  (*-- TRANSITION --------------------------------------------------------------------------------------------------------------*)
  IF (_CreateDir.bBusy = FALSE)
  THEN
    (*-- folder created => continue -----------------------------------------------------*)
    IF ( _CreateDir.bError = FALSE )
    THEN
      _WriteState:= E_TraceWriteStates.ScanFileStart;
      (*-- trace it -------------------------------------------------*)
// example: '11-000-0000-00-0, new folder created,  folder = D:/Traces/1979-01-09/'
      _Text:= '';
      _Text:= CONCAT(_Text, F_AddDividerToSisString(SubsystemRegistry.SubsystemName) );
      _Text:= CONCAT(_Text, ',  new folder created');
      _Text:= CONCAT(_Text, DebugTextBlocks.FOLDER);
      _Text:= CONCAT(_Text, _CreateDir.sPathName);
      Put( MsgType := E_DebugMsgType.INFO,
           Instance:= ADR(_Instance),
           Text    := ADR(_Text)  );
    (*-- folder already exists ----------------------------------------------------------*)
    ELSIF (    ( _CreateDir.nErrId = 16#070C )     // ADSERR_DEVICE_NOTFOUND
            OR ( _CreateDir.nErrId = 16#0723 )  )  // ADSERR_DEVICE_ACCESSDENIED
    THEN                                           // BKF-Flick: Änderung der ReturnCodes ab 4022.20
      _WriteState:= E_TraceWriteStates.ScanFileStart;
    (*-- error --------------------------------------------------------------------------*)
    ELSE
      _WriteState:= E_TraceWriteStates.Error;
    END_IF
  END_IF




(********************************************************************************************************************************)
(** prepare folder scan for existing files **************************************************************************************)
E_TraceWriteStates.ScanFileStart:
  (*-- ENTRY -------------------------------------------------------------------------------------------------------------------*)
  IF (_WriteStateLast <> _WriteState)
  THEN
    _WriteStateLast:= _WriteState;
    _WriteTime     := F_GetTimeMsTick();
    (*-----------------------------------------------------------------------------------*)
    _FileIndex     := 1;  (* Filenummerierung beginnt bei Eins *)
    _FileCheck.eCmd:= eEnumCmd_First;
  END_IF

  (*-- ACTION ------------------------------------------------------------------------------------------------------------------*)

  (*-- TRANSITION --------------------------------------------------------------------------------------------------------------*)
    _WriteState:= E_TraceWriteStates.ScanFileExists;




(********************************************************************************************************************************)
(** scan folder to check if files exist? ****************************************************************************************)
E_TraceWriteStates.ScanFileExists:
  (*-- ENTRY -------------------------------------------------------------------------------------------------------------------*)
  IF (_WriteStateLast <> _WriteState)
  THEN
    _WriteStateLast:= _WriteState;
    _WriteTime     := F_GetTimeMsTick();
    (*-- build file name with _FileIndex ------------------------------------------------*)
{warning disable C0139}
    M_BuildFileName();    _WriteFileName;
{warning restore C0139}
   (*-----------------------------------------------------------------------------------*)
    _FileCheck( bExecute:= FALSE );
    _FileCheck.sNetID   := '';  // local
//  _FileCheck.eCmd;   // maintain this value here 
    _FileCheck.bExecute := TRUE;
    _FileCheck.tTimeout := Tc2_System.DEFAULT_ADS_TIMEOUT;
    (*-----------------------------------------------------------------------------------*)
    DestStart:= ADR(_FileCheck.sPathName);
    DestEnd  := ADR(_FileCheck.sPathName) + SIZEOF(_FileCheck.sPathName);
    DestStart:= F_StringCopy( DestStart:= DestStart,  DestEnd:= DestEnd,  Source:= ADR(_WritePath)  );
    DestStart:= F_StringCopy( DestStart:= DestStart,  DestEnd:= DestEnd,  Source:= ADR(_WriteFileName)  );
  END_IF

  (*-- ACTION ------------------------------------------------------------------------------------------------------------------*)
  _FileCheck();

  (*-- TRANSITION --------------------------------------------------------------------------------------------------------------*)
  IF (_FileCheck.bBusy = FALSE)
  THEN
    _FileCheck.eCmd:= E_EnumCmdType.eEnumCmd_Next;
    (*-- error --------------------------------------------------------------------------*)
    IF ( _FileCheck.bError = TRUE )
    THEN
      _WriteState:= E_TraceWriteStates.Error;
    (*-- index does not exist => create & use -------------------------------------------*)
    ELSIF ( _FileCheck.bEOE = TRUE )
    THEN
      _WriteState:= E_TraceWriteStates.CreateOpen;
    (*-- found: but already too large => keep searching ---------------------------------*)
    ELSIF (    (_FileCheck.stFindFile.fileSize.dwLowPart)
            >= (_MaxFileSizeKB * DWORD#1024             )   ) (* kilo bytes => bytes *)
    THEN
      _WriteState:= E_TraceWriteStates.ScanFileCancel;
    (*-- found: smaller than max size => keep using -------------------------------------*)
    ELSE
      _WriteState:= E_TraceWriteStates.ScanFileAbort;
    END_IF
  END_IF




(********************************************************************************************************************************)
(** cancel scan *****************************************************************************************************************)
E_TraceWriteStates.ScanFileCancel:
  (*-- ENTRY -------------------------------------------------------------------------------------------------------------------*)
  IF (_WriteStateLast <> _WriteState)
  THEN
    _WriteStateLast:= _WriteState;
    _WriteTime     := F_GetTimeMsTick();
    (*-----------------------------------------------------------------------------------*)
    _FileCheck( bExecute:= FALSE );
    _FileCheck.sNetID   := '';  // local
//  _FileCheck.sPathName;  // maintain this value here 
    _FileCheck.eCmd     := E_EnumCmdType.eEnumCmd_Abort;
    _FileCheck.bExecute := TRUE;
    _FileCheck.tTimeout := Tc2_System.DEFAULT_ADS_TIMEOUT;
  END_IF

  (*-- ACTION ------------------------------------------------------------------------------------------------------------------*)
  _FileCheck();

  (*-- TRANSITION --------------------------------------------------------------------------------------------------------------*)
  IF (_FileCheck.bBusy = FALSE)
  THEN
    (*-- error --------------------------------------------------------------------------*)
    IF ( _FileCheck.bError = TRUE )
    THEN
      _WriteState:= E_TraceWriteStates.Error;
    (*-- cancellation successful --------------------------------------------------------*)
    ELSIF ( _FileCheck.bEOE = TRUE )
    THEN
      _FileIndex     := _FileIndex + 1;
      _FileCheck.eCmd:= eEnumCmd_First;
      _WriteState    := E_TraceWriteStates.ScanFileExists;
    (*-- keep searching -----------------------------------------------------------------*)
    ELSE
      _WriteStateLast:= E_TraceWriteStates.Initialization;  // Re-entry
    END_IF
  END_IF




(********************************************************************************************************************************)
(** cancel scan *****************************************************************************************************************)
E_TraceWriteStates.ScanFileAbort:
  (*-- ENTRY -------------------------------------------------------------------------------------------------------------------*)
  IF (_WriteStateLast <> _WriteState)
  THEN
    _WriteStateLast:= _WriteState;
    _WriteTime     := F_GetTimeMsTick();
    (*-----------------------------------------------------------------------------------*)
    _FileCheck( bExecute:= FALSE );
    _FileCheck.sNetID   := '';  // local
//  _FileCheck.sPathName;  // maintain this value here 
    _FileCheck.eCmd     := E_EnumCmdType.eEnumCmd_Abort;
    _FileCheck.bExecute := TRUE;
    _FileCheck.tTimeout := Tc2_System.DEFAULT_ADS_TIMEOUT;
  END_IF

  (*-- ACTION ------------------------------------------------------------------------------------------------------------------*)
  _FileCheck();

  (*-- TRANSITION --------------------------------------------------------------------------------------------------------------*)
  IF (_FileCheck.bBusy = FALSE)
  THEN
    (*-- error --------------------------------------------------------------------------*)
    IF    ( _FileCheck.bError = TRUE )
    THEN
      _WriteState:= E_TraceWriteStates.Error;
    (*-- cancellation successful --------------------------------------------------------*)
    ELSIF ( _FileCheck.bEOE = TRUE )
    THEN
      _WriteState:= E_TraceWriteStates.WaitForTrace;
    (*-- keep searching -----------------------------------------------------------------*)
    ELSE                                     
      _WriteStateLast:= E_TraceWriteStates.Initialization;  // Re-entry
    END_IF
  END_IF




(********************************************************************************************************************************)
(** create new file *************************************************************************************************************)
E_TraceWriteStates.CreateOpen:
  (*-- ENTRY -------------------------------------------------------------------------------------------------------------------*)
  IF (_WriteStateLast <> _WriteState)
  THEN
    _WriteStateLast:= _WriteState;
    _WriteTime     := F_GetTimeMsTick();
    (*-- build file name with _FileIndex ------------------------------------------------*)
{warning disable C0139}
    M_BuildFileName();    _WriteFileName;
{warning restore C0139}
    (*-----------------------------------------------------------------------------------*)
    _FileOpen( bExecute:= FALSE );
    _FileOpen.sNetId   := '';  // local
    _FileOpen.nMode    := ( FOPEN_MODEWRITE OR FOPEN_MODEPLUS OR FOPEN_MODEBINARY );
    _FileOpen.ePath    := E_OpenPath.PATH_GENERIC;          
    _FileOpen.bExecute := TRUE;
    _FileOpen.tTimeout := Tc2_System.DEFAULT_ADS_TIMEOUT;
    (*-----------------------------------------------------------------------------------*)
    DestStart:= ADR(_FileOpen.sPathName);
    DestEnd  := ADR(_FileOpen.sPathName) + SIZEOF(_FileOpen.sPathName);
    DestStart:= F_StringCopy( DestStart:= DestStart,  DestEnd:= DestEnd,  Source:= ADR(_WritePath)  );
    DestStart:= F_StringCopy( DestStart:= DestStart,  DestEnd:= DestEnd,  Source:= ADR(_WriteFileName)  );
  END_IF

  (*-- ACTION ------------------------------------------------------------------------------------------------------------------*)
  _FileOpen();

  (*-- TRANSITION --------------------------------------------------------------------------------------------------------------*)
  IF (_FileOpen.bBusy = FALSE)
  THEN
    (*-- File angelegt ------------------------------------------------------------------*)
    IF    ( _FileOpen.bError = FALSE )  
    THEN
      _Statistics.FileOpenCounter:= _Statistics.FileOpenCounter + 1;
      (*-----------------------------------------*)
      _Opened        := TRUE;
      _FileTimeOpened:= F_GetTimeMsTick();
      _WriteState    := E_TraceWriteStates.CreateHeader;
   (*-- folder doesn't exist (anymore) --------------------------------------------------*)
    ELSIF ( _FileOpen.nErrId = 16#070C )
    THEN
      _WriteState:= E_TraceWriteStates.StartWork;    
    (*-- error --------------------------------------------------------------------------*)
    ELSE
      _WriteState:= E_TraceWriteStates.Error;
    END_IF
  END_IF




(********************************************************************************************************************************)
(** write header ****************************************************************************************************************)
E_TraceWriteStates.CreateHeader:
  (*-- ENTRY -------------------------------------------------------------------------------------------------------------------*)
  IF (_WriteStateLast <> _WriteState)
  THEN
    _WriteStateLast:= _WriteState;
    _WriteTime     := F_GetTimeMsTick();
    (*-- create file header -------------------------------------------------------------*)
{warning disable C0139}
    M_CreateHeader();   _DataLength;
{warning restore C0139}
    (*-----------------------------------------------------------------------------------*)
    _FileWrite( bExecute:= FALSE );
    _FileWrite.sNetId    := '';  // local               
    _FileWrite.hFile     := _FileOpen.hFile;       
    _FileWrite.pWriteBuff:= ADR(_DataBuffer);
    _FileWrite.cbWriteLen:= _DataLength;
    _FileWrite.bExecute  := TRUE;
    _FileWrite.tTimeout  := Tc2_System.DEFAULT_ADS_TIMEOUT;
  END_IF

  (*-- ACTION ------------------------------------------------------------------------------------------------------------------*)
  _FileWrite();

  (*-- TRANSITION --------------------------------------------------------------------------------------------------------------*)
  IF (_FileWrite.bBusy = FALSE)
  THEN
    (*-- error --------------------------------------------------------------------------*)
    IF    ( _FileWrite.bError = TRUE )
    THEN
      _WriteState:= E_TraceWriteStates.Error;
    (*-- writing successful -------------------------------------------------------------*)
    ELSE
      _WriteState:= E_TraceWriteStates.CreateClose;
    END_IF
  END_IF




(********************************************************************************************************************************)
(** close new file **************************************************************************************************************)
E_TraceWriteStates.CreateClose:
  (*-- ENTRY -------------------------------------------------------------------------------------------------------------------*)
  IF (_WriteStateLast <> _WriteState)
  THEN
    _WriteStateLast:= _WriteState;
    _WriteTime     := F_GetTimeMsTick();
    (*-----------------------------------------------------------------------------------*)
    _FileClose( bExecute:= FALSE );
    _FileClose.sNetId  := '';   // local
    _FileClose.hFile   := _FileOpen.hFile;
    _FileClose.bExecute:= TRUE;
    _FileClose.tTimeout:= Tc2_System.DEFAULT_ADS_TIMEOUT;
  END_IF

  (*-- ACTION ------------------------------------------------------------------------------------------------------------------*)
  _FileClose();

  (*-- TRANSITION --------------------------------------------------------------------------------------------------------------*)
  IF (_FileClose.bBusy = FALSE)
  THEN
    _PlcRestarted:= FALSE;
    _Opened      := FALSE;
    (*-- calculate maximum file open time -----------------------------------------------*)
    _Statistics.MaxFileOpenTime:= MAX( _Statistics.MaxFileOpenTime, F_GetTimeMsDiff(_FileTimeOpened)  );
    (*-- error --------------------------------------------------------------------------*)
    IF    ( _FileClose.bError = TRUE )
    THEN
      _WriteState:= E_TraceWriteStates.Error;
    (*-- closing successful -------------------------------------------------------------*)
    ELSE
      _WriteState:= E_TraceWriteStates.WaitForTrace;
    END_IF
  END_IF




(********************************************************************************************************************************)
(** inhibit time (currently not used) *******************************************************************************************)
E_TraceWriteStates.WaitLocked:
  (*-- ENTRY -------------------------------------------------------------------------------------------------------------------*)
  IF (_WriteStateLast <> _WriteState)
  THEN
    _WriteStateLast:= _WriteState;
    _WriteTime     := F_GetTimeMsTick();
    (*-----------------------------------------------------------------------------------*)
  END_IF

  (*-- ACTION ------------------------------------------------------------------------------------------------------------------*)

  (*-- TRANSITION --------------------------------------------------------------------------------------------------------------*)
  (*-- (still) too many traces to be written -> skip inhibit time -----------------------*)
  IF (_FifoFillLevel >= 256)
  THEN
    _WriteState:= E_TraceWriteStates.WaitForTrace;
  (*-- inhibit time over ----------------------------------------------------------------*)
  ELSIF (F_GetTimeMsDiff(_WriteTime) >= LOCKTIME)
  THEN
    _WriteState:= E_TraceWriteStates.WaitForTrace;
  (*-- working folder dissapeared -------------------------------------------------------*)
  ELSIF (_Active = FALSE)
  THEN
    _WriteState:= E_TraceWriteStates.WaitFolder;
  END_IF




(********************************************************************************************************************************)
(** idle -> wait for traces to write ********************************************************************************************)
E_TraceWriteStates.WaitForTrace:
  (*-- ENTRY -------------------------------------------------------------------------------------------------------------------*)
  IF (_WriteStateLast <> _WriteState)
  THEN
    _WriteStateLast:= _WriteState;
    _WriteTime     := F_GetTimeMsTick();
    (*-----------------------------------------------------------------------------------*)
  END_IF

  (*-- ACTION ------------------------------------------------------------------------------------------------------------------*)

  (*-- TRANSITION --------------------------------------------------------------------------------------------------------------*)
  (*-- traces to write available --------------------------------------------------------*)
  IF (_FifoFillLevel <> 0)
  THEN
//  IF ( _FileIndex <> 1 ) 
//  THEN
//     => check if file-one (still) exists
//  ELSE
    _FileCheck.eCmd:= E_EnumCmdType.eEnumCmd_First;
    _WriteState    := E_TraceWriteStates.FileSizeExists;
  (*-- working folder dissapeared -------------------------------------------------------*)
  ELSIF (_Active = FALSE)
  THEN
    _WriteState:= E_TraceWriteStates.WaitFolder;
  END_IF




(********************************************************************************************************************************)
(** check if current file (_FileIndex) still exists and if it's (already) too large *********************************************)
E_TraceWriteStates.FileSizeExists:
  (*-- ENTRY -------------------------------------------------------------------------------------------------------------------*)
  IF (_WriteStateLast <> _WriteState)
  THEN
    _WriteStateLast:= _WriteState;
    _WriteTime     := F_GetTimeMsTick();
    (*-----------------------------------------------------------------------------------*)
    _FileCheck( bExecute:= FALSE );
    _FileCheck.sNetID   := '';   // local
//  _FileCheck.eCmd;   (* nicht beschreiben *)
    _FileCheck.bExecute := TRUE;
    _FileCheck.tTimeout := Tc2_System.DEFAULT_ADS_TIMEOUT;
    (*-----------------------------------------------------------------------------------*)
    DestStart:= ADR(_FileCheck.sPathName);
    DestEnd  := ADR(_FileCheck.sPathName) + SIZEOF(_FileCheck.sPathName);
    DestStart:= F_StringCopy( DestStart:= DestStart,  DestEnd:= DestEnd,  Source:= ADR(_WritePath)  );
    DestStart:= F_StringCopy( DestStart:= DestStart,  DestEnd:= DestEnd,  Source:= ADR(_WriteFileName)  );
  END_IF

  (*-- ACTION ------------------------------------------------------------------------------------------------------------------*)
  _FileCheck();

  (*-- TRANSITION --------------------------------------------------------------------------------------------------------------*)
  IF (_FileCheck.bBusy = FALSE)
  THEN
    (*-- error --------------------------------------------------------------------------*)
    IF    (_FileCheck.bError = TRUE)
    THEN
      _WriteState:= E_TraceWriteStates.Error;
    (*-- doesnt exists (anymore) => rescan ----------------------------------------------*)
    ELSIF (_FileCheck.bEOE = TRUE)
    THEN
      _WriteState:= E_TraceWriteStates.ScanFileStart;
    (*-- exists: => use it --------------------------------------------------------------*)
    ELSE
      _FileSize  := (        DWORD_TO_ULINT(_FileCheck.stFindFile.fileSize.dwLowPart )
                      OR SHL(DWORD_TO_ULINT(_FileCheck.stFindFile.fileSize.dwHighPart), 32)  );
      (*-- maximal file size exceeded -----------*)
      IF (    (_FileSize (* KiloBytes => Bytes *) )
           >= (_MaxFileSizeKB * ULINT#1024        )   )  THEN   _WriteState:= E_TraceWriteStates.FileSizeCancel;  // start over with new file index
      ELSE                                                      _WriteState:= E_TraceWriteStates.FileSizeAbort;   // use this file again
      END_IF
    END_IF
  END_IF




(********************************************************************************************************************************)
(** cancel file size/exist check and use this ***********************************************************************************)
E_TraceWriteStates.FileSizeAbort:
  (*-- ENTRY -------------------------------------------------------------------------------------------------------------------*)
  IF (_WriteStateLast <> _WriteState)
  THEN
    _WriteStateLast:= _WriteState;
    _WriteTime     := F_GetTimeMsTick();
    (*-----------------------------------------------------------------------------------*)
    _FileCheck( bExecute:= FALSE );
    _FileCheck.sNetID   := '';   // local
//  _FileCheck.sPathName;  remain value
    _FileCheck.eCmd     := E_EnumCmdType.eEnumCmd_Abort;
    _FileCheck.bExecute := TRUE;
    _FileCheck.tTimeout := Tc2_System.DEFAULT_ADS_TIMEOUT;
  END_IF

  (*-- ACTION ------------------------------------------------------------------------------------------------------------------*)
  _FileCheck();

  (*-- TRANSITION --------------------------------------------------------------------------------------------------------------*)
  IF ( _FileCheck.bBusy = FALSE )
  THEN
    (*-- error --------------------------------------------------------------------------*)
    IF    (_FileCheck.bError = TRUE)
    THEN
      _WriteState:= E_TraceWriteStates.Error;
    (*-- finished -----------------------------------------------------------------------*)
    ELSIF (_FileCheck.bEOE = TRUE)
    THEN
      _WriteState:= E_TraceWriteStates.OpenAppend;
    (*-- keep searching -----------------------------------------------------------------*)
    ELSE
      _WriteStateLast:= E_TraceWriteStates.Initialization;  // Re-entry
    END_IF
  END_IF



(********************************************************************************************************************************)
(** cancel file size/exist check due to file size already too large *************************************************************)
E_TraceWriteStates.FileSizeCancel:
  (*-- ENTRY -------------------------------------------------------------------------------------------------------------------*)
  IF (_WriteStateLast <> _WriteState)
  THEN
    _WriteStateLast:= _WriteState;
    _WriteTime     := F_GetTimeMsTick();
    (*-----------------------------------------------------------------------------------*)
    _FileCheck( bExecute:= FALSE );
    _FileCheck.sNetID   := '';   // local
//  _FileCheck.sPathName;  remain value
    _FileCheck.eCmd     := E_EnumCmdType.eEnumCmd_Abort;
    _FileCheck.bExecute := TRUE;
    _FileCheck.tTimeout := Tc2_System.DEFAULT_ADS_TIMEOUT;
  END_IF

  (*-- ACTION ------------------------------------------------------------------------------------------------------------------*)
  _FileCheck();

  (*-- TRANSITION --------------------------------------------------------------------------------------------------------------*)
  IF ( _FileCheck.bBusy = FALSE )
  THEN
    (*-- error --------------------------------------------------------------------------*)
    IF    (_FileCheck.bError = TRUE)
    THEN
      _WriteState:= E_TraceWriteStates.Error;
    (*-- finished -----------------------------------------------------------------------*)
    ELSIF (_FileCheck.bEOE = TRUE)
    THEN
      _FileIndex := _FileIndex + 1;
      _WriteState:= E_TraceWriteStates.CreateOpen;
    (*-- keep searching -----------------------------------------------------------------*)
    ELSE
      _WriteStateLast:= E_TraceWriteStates.Initialization;  // Re-entry
    END_IF
  END_IF




(********************************************************************************************************************************)
(** open file to write/append ***************************************************************************************************)
E_TraceWriteStates.OpenAppend:
  (*-- ENTRY -------------------------------------------------------------------------------------------------------------------*)
  IF (_WriteStateLast <> _WriteState)
  THEN
    _WriteStateLast:= _WriteState;
    _WriteTime     := F_GetTimeMsTick();
    (*-----------------------------------------------------------------------------------*)
    _FileOpen( bExecute:= FALSE );
    _FileOpen.sNetId   := '';   // local
    _FileOpen.nMode    := ( FOPEN_MODEAPPEND OR FOPEN_MODEBINARY );                                
    _FileOpen.ePath    := E_OpenPath.PATH_GENERIC;          
    _FileOpen.bExecute := TRUE;
    _FileOpen.tTimeout := Tc2_System.DEFAULT_ADS_TIMEOUT;
    (*-----------------------------------------------------------------------------------*)
    DestStart:= ADR(_FileOpen.sPathName);
    DestEnd  := ADR(_FileOpen.sPathName) + SIZEOF(_FileOpen.sPathName);
    DestStart:= F_StringCopy( DestStart:= DestStart,  DestEnd:= DestEnd,  Source:= ADR(_WritePath)  );
    DestStart:= F_StringCopy( DestStart:= DestStart,  DestEnd:= DestEnd,  Source:= ADR(_WriteFileName)  );
  END_IF

  (*-- ACTION ------------------------------------------------------------------------------------------------------------------*)
  _FileOpen();

  (*-- TRANSITION --------------------------------------------------------------------------------------------------------------*)
  IF ( _FileOpen.bBusy = FALSE )
  THEN
    (*-- file opened --------------------------------------------------------------------*)
    IF    ( _FileOpen.bError = FALSE )  
    THEN
      _Statistics.FileOpenCounter:= _Statistics.FileOpenCounter + 1;
      _FileTimeOpened            := F_GetTimeMsTick();
      _Opened                    := TRUE;
      (*-----------------------------------------*)
      IF (_PlcRestarted = TRUE) THEN   _WriteState:= E_TraceWriteStates.WriteDivider;
      ELSE                             _WriteState:= E_TraceWriteStates.WriteData;
      END_IF
    (*-- folder doesn't exist (anymore) -------------------------------------------------*)
    ELSIF ( _FileOpen.nErrId = 16#070C )
    THEN
      _WriteState:= E_TraceWriteStates.StartWork;    
    (*-- error --------------------------------------------------------------------------*)
    ELSE
      _WriteState:= E_TraceWriteStates.Error;
    END_IF
  END_IF




(********************************************************************************************************************************)
(** add plc restart divider *****************************************************************************************************)
E_TraceWriteStates.WriteDivider:
  (*-- ENTRY -------------------------------------------------------------------------------------------------------------------*)
  IF (_WriteStateLast <> _WriteState)
  THEN
    _WriteStateLast:= _WriteState;
    _WriteTime     := F_GetTimeMsTick();
    (*-- create plc divider -------------------------------------------------------------*)
{warning disable C0139}
    M_CreatePlcDivider();   _DataLength;
{warning restore C0139}
    (*-----------------------------------------------------------------------------------*)
    _FileWrite( bExecute:= FALSE );
    _FileWrite.sNetId    := '';  // local               
    _FileWrite.hFile     := _FileOpen.hFile;       
    _FileWrite.pWriteBuff:= ADR(_DataBuffer);
    _FileWrite.cbWriteLen:= _DataLength;
    _FileWrite.bExecute  := TRUE;
    _FileWrite.tTimeout  := Tc2_System.DEFAULT_ADS_TIMEOUT;
  END_IF

  (*-- ACTION ------------------------------------------------------------------------------------------------------------------*)
  _FileWrite();

  (*-- TRANSITION --------------------------------------------------------------------------------------------------------------*)
  IF (_FileWrite.bBusy = FALSE)
  THEN
    _PlcRestarted:= FALSE;
    _FileSize    := _FileSize + _FileWrite.cbWrite;
    (*-- error --------------------------------------------------------------------------*)
    IF    (_FileWrite.bError = TRUE)
    THEN
      _WriteState:= E_TraceWriteStates.CloseOpenTime;
    (*-- writing successful -------------------------------------------------------------*)
    ELSE
      _WriteState:= E_TraceWriteStates.WriteData;
    END_IF
  END_IF




(********************************************************************************************************************************)
(** write trace lines ***********************************************************************************************************)
E_TraceWriteStates.WriteData:
  (*-- ENTRY -------------------------------------------------------------------------------------------------------------------*)
  IF (_WriteStateLast <> _WriteState)
  THEN
    _WriteStateLast:= _WriteState;
    _WriteTime     := F_GetTimeMsTick();
    (*-- create data --------------------------------------------------------------------*)
{warning disable C0139}
    _DataDateChanged:= M_CreateData();   _DataLength;
    (*-----------------------------------------------------------------------------------*)
    _FileWrite( bExecute:= FALSE );
    _FileWrite.sNetId    := '';  // local               
    _FileWrite.hFile     := _FileOpen.hFile;       
    _FileWrite.pWriteBuff:= ADR(_DataBuffer);
    _FileWrite.cbWriteLen:= _DataLength;
    _FileWrite.bExecute  := TRUE;
    _FileWrite.tTimeout  := Tc2_System.DEFAULT_ADS_TIMEOUT;
{warning restore C0139}
  END_IF

  (*-- ACTION ------------------------------------------------------------------------------------------------------------------*)
  _FileWrite();

  (*-- TRANSITION --------------------------------------------------------------------------------------------------------------*)
  IF ( _FileWrite.bBusy = FALSE )
  THEN
    _FileSize:= _FileSize + _FileWrite.cbWrite;
    (*-- error --------------------------------------------------------------------------*)
    IF    (_FileWrite.bError = TRUE)
    THEN
      _WriteState:= E_TraceWriteStates.CloseOpenTime;
    (*-- trace date changed -> new date folder ------------------------------------------*)
    ELSIF (_DataDateChanged = TRUE)
    THEN  (* new file/folder for new day *)
      _WriteState:= E_TraceWriteStates.EofDate;
    (*-- maximum file size exceeded -----------------------------------------------------*)
    ELSIF (    (_FileSize (* KiloBytes => Bytes *) )
            >= (_MaxFileSizeKB * ULINT#1024        )   )
    THEN  (* start over with new file index *)
      _WriteState:= E_TraceWriteStates.EofSize;
    (*-- maximum file open time exceeded (flush) ----------------------------------------*)
    ELSIF (F_GetTimeMsDiff(_FileTimeOpened) >= MAX_FILEOPEN_TIME)
    THEN  (* close file and re-open it => file flush *)
      _WriteState:= E_TraceWriteStates.CloseOpenTime;
    (*-- more to write? -----------------------------------------------------------------*)
    ELSIF (_FifoFillLevel <> 0)
    THEN
      _WriteStateLast:= E_TraceWriteStates.Initialization;  // Re-entry
    (*-- no traces to write anymore -> close & wait -------------------------------------*)
    ELSE
      _WriteState:= E_TraceWriteStates.CloseOpenTime;
    END_IF
  END_IF




(********************************************************************************************************************************)
(** close due to max open time exceeded *****************************************************************************************)
E_TraceWriteStates.CloseOpenTime:
  (*-- ENTRY -------------------------------------------------------------------------------------------------------------------*)
  IF (_WriteStateLast <> _WriteState)
  THEN
    _WriteStateLast:= _WriteState;
    _WriteTime     := F_GetTimeMsTick();
    (*-----------------------------------------------------------------------------------*)
    _FileClose( bExecute:= FALSE );
    _FileClose.sNetId  := '';  // local
    _FileClose.hFile   := _FileOpen.hFile;
    _FileClose.bExecute:= TRUE;
    _FileClose.tTimeout:= Tc2_System.DEFAULT_ADS_TIMEOUT;
  END_IF

  (*-- ACTION ------------------------------------------------------------------------------------------------------------------*)
  _FileClose();

  (*-- TRANSITION --------------------------------------------------------------------------------------------------------------*)
  IF (_FileClose.bBusy = FALSE)
  THEN
    _Opened:= FALSE;
    (*-- calculate maximum file open time -----------------------------------------------*)
    _Statistics.MaxFileOpenTime:= MAX( _Statistics.MaxFileOpenTime, F_GetTimeMsDiff(_FileTimeOpened)  );
    (*-- error --------------------------------------------------------------------------*)
    IF    (_FileClose.bError = TRUE)
    THEN
      _WriteState:= E_TraceWriteStates.Error;
    (*-- closing successful -------------------------------------------------------------*)
    ELSE
      _WriteState:= E_TraceWriteStates.WaitLocked;
    END_IF
  END_IF




(********************************************************************************************************************************)
(** add eof due max file size exceeded ******************************************************************************************)
E_TraceWriteStates.EofSize:
  (*-- ENTRY -------------------------------------------------------------------------------------------------------------------*)
  IF (_WriteStateLast <> _WriteState)
  THEN
    _WriteStateLast:= _WriteState;
    _WriteTime     := F_GetTimeMsTick();
    (*-- create eof ---------------------------------------------------------------------*)
{warning disable C0139}
    M_CreateEof();   _DataLength;
{warning restore C0139}
    (*-----------------------------------------------------------------------------------*)
    _FileWrite( bExecute:= FALSE );
    _FileWrite.sNetId    := '';  // local               
    _FileWrite.hFile     := _FileOpen.hFile;       
    _FileWrite.pWriteBuff:= ADR(_DataBuffer);
    _FileWrite.cbWriteLen:= _DataLength;
    _FileWrite.bExecute  := TRUE;
    _FileWrite.tTimeout  := Tc2_System.DEFAULT_ADS_TIMEOUT;
  END_IF

  (*-- ACTION ------------------------------------------------------------------------------------------------------------------*)
  _FileWrite();

  (*-- TRANSITION --------------------------------------------------------------------------------------------------------------*)
  IF (_FileWrite.bBusy = FALSE)
  THEN
    _FileSize  := _FileSize + _FileWrite.cbWrite;
    _WriteState:= E_TraceWriteStates.CloseSize;
  END_IF




(********************************************************************************************************************************)
(** close due to max file size exceeded *****************************************************************************************)
E_TraceWriteStates.CloseSize:
  (*-- ENTRY -------------------------------------------------------------------------------------------------------------------*)
  IF (_WriteStateLast <> _WriteState)
  THEN
    _WriteStateLast:= _WriteState;
    _WriteTime     := F_GetTimeMsTick();
    (*-----------------------------------------------------------------------------------*)
    _FileClose( bExecute:= FALSE );
    _FileClose.sNetId  := '';  // local
    _FileClose.hFile   := _FileOpen.hFile;
    _FileClose.bExecute:= TRUE;
    _FileClose.tTimeout:= Tc2_System.DEFAULT_ADS_TIMEOUT;
  END_IF

  (*-- ACTION ------------------------------------------------------------------------------------------------------------------*)
  _FileClose();

  (*-- TRANSITION --------------------------------------------------------------------------------------------------------------*)
  IF (_FileClose.bBusy = FALSE)
  THEN
    _FileIndex:= _FileIndex + 1;
    _Opened   := FALSE;
    (*-- calculate maximum file open time -----------------------------------------------*)
    _Statistics.MaxFileOpenTime:= MAX( _Statistics.MaxFileOpenTime, F_GetTimeMsDiff(_FileTimeOpened)  );
    (*-- error --------------------------------------------------------------------------*)
    IF    (_FileClose.bError = TRUE)
    THEN
      _WriteState:= E_TraceWriteStates.Error;
    (*-- closing successful -------------------------------------------------------------*)
    ELSE
      _WriteState:= E_TraceWriteStates.CreateOpen;
    END_IF
  END_IF




(********************************************************************************************************************************)
(** add eof due to new date *****************************************************************************************************)
E_TraceWriteStates.EofDate:
  (*-- ENTRY -------------------------------------------------------------------------------------------------------------------*)
  IF (_WriteStateLast <> _WriteState)
  THEN
    _WriteStateLast:= _WriteState;
    _WriteTime     := F_GetTimeMsTick();
    (*-- create eof ---------------------------------------------------------------------*)
{warning disable C0139}
    M_CreateEof();   _DataLength;
{warning restore C0139}
    (*-----------------------------------------------------------------------------------*)
    _FileWrite( bExecute:= FALSE );
    _FileWrite.sNetId    := '';  // local               
    _FileWrite.hFile     := _FileOpen.hFile;       
    _FileWrite.pWriteBuff:= ADR(_DataBuffer);
    _FileWrite.cbWriteLen:= _DataLength;
    _FileWrite.bExecute  := TRUE;
    _FileWrite.tTimeout  := Tc2_System.DEFAULT_ADS_TIMEOUT;
  END_IF

  (*-- ACTION ------------------------------------------------------------------------------------------------------------------*)
  _FileWrite();

  (*-- TRANSITION --------------------------------------------------------------------------------------------------------------*)
  IF (_FileWrite.bBusy = FALSE)
  THEN
    _FileSize  := _FileSize + _FileWrite.cbWrite;
    _WriteState:= E_TraceWriteStates.CloseDate;
  END_IF




(********************************************************************************************************************************)
(** close due to new date *******************************************************************************************************)
E_TraceWriteStates.CloseDate:
  (*-- ENTRY -------------------------------------------------------------------------------------------------------------------*)
  IF (_WriteStateLast <> _WriteState)
  THEN
    _WriteStateLast:= _WriteState;
    _WriteTime     := F_GetTimeMsTick();
    (*-----------------------------------------------------------------------------------*)
    _FileClose( bExecute:= FALSE );
    _FileClose.sNetId  := '';  // local
    _FileClose.hFile   := _FileOpen.hFile;
    _FileClose.bExecute:= TRUE;
    _FileClose.tTimeout:= Tc2_System.DEFAULT_ADS_TIMEOUT;
  END_IF

  (*-- ACTION ------------------------------------------------------------------------------------------------------------------*)
  _FileClose();

  (*-- TRANSITION --------------------------------------------------------------------------------------------------------------*)
  IF (_FileClose.bBusy = FALSE)
  THEN
    _Opened:= FALSE;
    (*-- calculate maximum file open time -----------------------------------------------*)
    _Statistics.MaxFileOpenTime:= MAX( _Statistics.MaxFileOpenTime, F_GetTimeMsDiff(_FileTimeOpened)  );
    (*-- error --------------------------------------------------------------------------*)
    IF    (_FileClose.bError = TRUE)
    THEN
      _WriteState:= E_TraceWriteStates.Error;
    (*-- closing successful -------------------------------------------------------------*)
    ELSE
      _WriteState:= E_TraceWriteStates.HddUsage;
    END_IF
  END_IF




(********************************************************************************************************************************)
(** read current hdd usage ******************************************************************************************************)
E_TraceWriteStates.HddUsage:
  (*-- ENTRY -------------------------------------------------------------------------------------------------------------------*)
  IF (_WriteStateLast <> _WriteState)
  THEN
    _WriteStateLast:= _WriteState;
    _WriteTime     := F_GetTimeMsTick();
    (*-----------------------------------------------------------------------------------*)
    _HddUsage.Start( Drive:= _MainFolder );  // use drive letter from main folder
  END_IF

  (*-- ACTION ------------------------------------------------------------------------------------------------------------------*)

  (*-- TRANSITION --------------------------------------------------------------------------------------------------------------*)
  IF (_HddUsage.Busy = FALSE)
  THEN
    _HddUsageCount:= _HddUsageCount + 1;
    _HddStateLast := E_TraceHddUsageStates.Initialization;  // force re-entry and write message
    (*-------------------------------------------*)
    _WriteState:= E_TraceWriteStates.StartWork;
  END_IF




(********************************************************************************************************************************)
(** unknown *********************************************************************************************************************)
ELSE
  _WriteState:= E_TraceWriteStates.Initialization;
END_CASE




(********************************************************************************************************************************)
(** done ************************************************************************************************************************)
END_METHOD

// maximum file size in kilobytes
{attribute 'monitoring' := 'call'}
PROPERTY PUBLIC MaxFileSizeKB : WORD
GET
MaxFileSizeKB:= _MaxFileSizeKB;
END_GET
SET
_MaxFileSizeKB:= MaxFileSizeKB;
END_SET
END_PROPERTY

// HI = file is currently open
{attribute 'monitoring' := 'call'}
PROPERTY PUBLIC Opened : BOOL
GET
Opened:= _Opened;
END_GET
END_PROPERTY

// puts a new trace line into the current file
METHOD PUBLIC Put

(********************************************************************************************************************************)
VAR_INPUT
  MsgType               : E_DebugMsgType                   := E_DebugMsgType.ERROR;
  Instance              : POINTER TO BYTE                  := 0;     // pointer to string
  Text                  : POINTER TO BYTE                  := 0;     // pointer to string
END_VAR

(********************************************************************************************************************************)
VAR
  Entry                 : POINTER TO FB_TraceEntry         := 0;
END_VAR

(********************************************************************************************************************************)
(** check inputs ****************************************************************************************************************)
IF (Text = 0)
THEN
  RETURN;
END_IF




(********************************************************************************************************************************)
(** enough hdd space? ***********************************************************************************************************)
IF (_HddTooFull = TRUE)
THEN
  _HddFullMissed:= _HddFullMissed + 1;
  RETURN;
END_IF




(********************************************************************************************************************************)
(** fb ready? *******************************************************************************************************************)
IF (System.fbSystemTime.TIMESTR.wYear = 0)
THEN
  _Diag_InvalidDate:= _Diag_InvalidDate + 1;
  RETURN;
END_IF




(********************************************************************************************************************************)
(** space in fifo available? ****************************************************************************************************)
IF (_FifoFillLevel >= FIFO_SIZE)
THEN
  _Diag_FifoFull:= _Diag_FifoFull + 1;
  RETURN;
END_IF




(********************************************************************************************************************************)
(** create entry ****************************************************************************************************************)
Entry:= __NEW( FB_TraceEntry( DateTime   := System.fbSystemTime.TIMESTR,
                              TaskCounter:= _TaskCounter + 1,
                             xMsgType    := MsgType,
                             xInstance   := Instance,  // leading x in the name:
                              Text       := Text  ) ); // Beckhoff SUPPORTCH-29439
IF   (Entry        = 0)      THEN  _Diag_NoMemory:= _Diag_NoMemory + 1;  RETURN;
ELSIF(Entry^.Valid = FALSE)  THEN  _Diag_NoEntry := _Diag_NoEntry  + 1;  __DELETE(Entry);  RETURN;
END_IF

_TaskCounter:= _TaskCounter + 1;





(********************************************************************************************************************************)
(** put into fifo ***************************************************************************************************************)
_Fifo[_FifoInput]:= Entry;

_FifoInput:= _FifoInput + 1;
IF(_FifoInput >= FIFO_SIZE)
THEN
  _FifoInput:= 0;
END_IF

_FifoFillLevel:= _FifoFillLevel + 1;




(********************************************************************************************************************************)
(** update statistics ***********************************************************************************************************)
_Statistics.PutCounter      := _Statistics.PutCounter  + 1;
_Statistics.MaxFifoFillLevel:= MAX(_Statistics.MaxFifoFillLevel, _FifoFillLevel);




(********************************************************************************************************************************)
(** done ************************************************************************************************************************)
END_METHOD

// diagnosis & statisticals
{attribute 'monitoring' := 'call'}
PROPERTY PUBLIC Statistics : I_TraceHandlerStatistics
GET
Statistics:= _Statistics;
END_GET
END_PROPERTY

END_FUNCTION_BLOCK

(* stored: Version 1.1.0.1, ProductVersion 3.1.4024.4
   POU FB_TraceHandler: Id {3890a7ed-527c-4f6c-96a1-16982dfd8078}, SpecialFunc None
   Folder _internal: Id {c5145b27-8783-45c2-aed9-32baf585f4e3}
   Folder Methods: Id {1b117e47-6bfc-478a-8c70-073dd0ec4d53}
   Folder Properties: Id {fa1dee63-984d-462e-9bc3-d37e0874f870}
   Method Clear: Id {48b7b36e-ba2d-431c-a64a-01282951e7eb}
   Property Enable: Id {e0744883-537a-445c-872c-edfa035389a1}
   Get Get: Id {54a5c298-ac89-42c6-9756-b9496a8e1c39}
   Set Set: Id {6d238f31-1482-427b-99a7-cc9ae9dbc7f3}
   Method FB_exit: Id {8f532351-763f-4b76-8185-30859ec27a99}
   Method FB_init: Id {3508e532-e4bc-4cb5-9ee0-2517077e334a}
   Property Folder: Id {66c8f564-b69a-4e81-bc93-da25321a68d9}
   Get Get: Id {72d936d2-6b94-478b-bef6-c0924e425507}
   Set Set: Id {3a26c8c8-e784-42e4-ba35-0e2a41a0144a}
   Property HddUsage: Id {4c18a9fc-e734-43d0-8a56-52ba2f642d30}
   Get Get: Id {02a75c85-74cc-455b-b53c-fc1b172e070c}
   Method M_BuildFileName: Id {1ecd50bb-b1f1-4708-8c7e-314d58ff6779}
   Method M_CreateData: Id {18a650e2-4f51-4483-ae60-e6f91bb07b68}
   Method M_CreateEof: Id {637a1451-9874-4b27-86f1-1ed3c754f694}
   Method M_CreateHeader: Id {d1cc4121-f79a-45b7-895f-48f85bf783fe}
   Method M_CreatePlcDivider: Id {6d1fdd25-f6ab-43e8-a86d-f3432d14430a}
   Method M_RunCheck: Id {b8196444-94e0-454c-8862-e3abc8510994}
   Method M_RunDelete: Id {0e496b6a-69e1-4e77-8a08-52e23a8bcf7c}
   Method M_RunHddUsage: Id {b3fef0c1-5681-43b3-a8ff-57e405e5781c}
   Method M_RunWrite: Id {a392f093-5d18-490d-bbb7-0e5bd0e5e96c}
   Property MaxFileSizeKB: Id {1d4164e0-a4af-4d8c-a3a2-e235dae19903}
   Get Get: Id {2af74c19-ff28-4e7f-910a-845c33d12fee}
   Set Set: Id {eca2550f-655d-4484-827b-dc6bceef6ff7}
   Property Opened: Id {617ecbad-aa95-481c-a979-34e8e62c38de}
   Get Get: Id {90665bb4-caf1-4117-a5b0-042d9f5eb61d}
   Method Put: Id {67d6dd9d-f152-4b22-9130-6bac5fcc1978}
   Property Statistics: Id {88415d1b-8357-46eb-91be-3330e3ce453d}
   Get Get: Id {75d4b5c9-f52e-4f03-9bed-3fef83ad743c} *)
